PROGRAM P_Demo_FB_DMXGetSensorValue
VAR
    fbGetSensorVal    : FB_DMXGetSensorValue;         // 读传感器当前值
    stDmxCmdBuffer    : ST_DMXCommandBuffer;          // 与通讯 FB 共用
    wTargetManufId    : WORD := 16#4241;              // 目标灯具厂商 ID
    dwTargetDeviceId  : DWORD := 16#12131415;         // 目标灯具设备 ID
    byTargetPort      : BYTE := 0;                    // 根设备通道 0
    bySensorIndex     : BYTE := 0;                    // 第一个传感器（如温度）
    bDoRead           : BOOL := FALSE;                // 在线给一次上升沿触发
    bBusy             : BOOL;
    bError            : BOOL;
    udiErrId          : UDINT;
    stSensorVal       : ST_DMXSensorValue;            // 传感器值结构
END_VAR

// ============================================================
// Tc2_DMX.FB_DMXGetSensorValue 演示程序
// ============================================================
// 场景：灯具过温保护监控：周期读每盏灯温度传感器当前值，超阈值时 PLC 降功率或报警防过热。
// 价值：把灯具内部传感器实时值接入 PLC，实现基于真实物理量的保护与预测性维护。
// 验证：设 bySensorIndex:=0，给 bDoRead 一次上升沿 -> bBusy 短暂 TRUE -> 回 FALSE 后 stSensorVal 含当前值/最低值/最高值；配合 FB_DMXGetSensorDefinition 的单位换算成实际温度。
// 验证步骤：
//   1. 右键 PLC 项目下 POUs 文件夹 → Add → Existing Item → 选本 .TcPOU 文件
//   2. 引用 Tc2_DMX；同项目里放一个 FB_EL6851CommunicationEx 实例并共用 stDmxCmdBuffer（非 CycleMode）
//   3. 编译 → 登录 → 运行；按上方『验证』行在线给上升沿观察
// ============================================================

fbGetSensorVal(
    bStart                     := bDoRead,
    wDestinationManufacturerId := wTargetManufId,
    dwDestinationDeviceId      := dwTargetDeviceId,
    byPortId                   := byTargetPort,
    bySensorNumber             := bySensorIndex,
    dwOptions                  := 0,
    stCommandBuffer            := stDmxCmdBuffer,
    bBusy                      => bBusy,
    bError                     => bError,
    udiErrorId                 => udiErrId,
    stDMXSensorValue           => stSensorVal
);

END_PROGRAM

(* stored: Version 1.1.0.1, ProductVersion 3.1.4024.5
   POU P_Demo_FB_DMXGetSensorValue: Id {59762c9d-3198-58da-8eb9-e377ce21e68e}, SpecialFunc None *)
